// TIA Portal V16 export
// export: Created 2021-05-26T11:52:20.4679545Z, ExportSetting WithDefaults, DisplayName Totally Integrated Automation Portal, DisplayVersion V16 Update 4, DisplayName TIA Portal Version Control Interface, DisplayVersion V16 Update 2, DisplayName TIA Portal Openness, DisplayVersion V16 Update 4, DisplayName STEP 7 Professional, DisplayVersion V16 Update 4, DisplayName STEP 7 Safety, DisplayVersion V16, DisplayName WinCC Advanced, DisplayVersion V16 Update 4
DATA_BLOCK "DB_BC"   // DB10
{ S7_Optimized_Access := 'FALSE'; DB_Accessible_From_OPC_UA := 'FALSE' }
VERSION : 0.1
// stored: AutoNumber false, DBAccessibleFromOPCUA false, IsOnlyStoredInLoadMemory false, IsWriteProtectedInAS false
   VAR
      Spare0 : Byte;
      cmdRegLo : Bool;
      cmdBCRstHi : Bool;
      res_b1_2 : Bool;
      res_b1_3 : Bool;
      res_b1_4 : Bool;
      res_b1_5 : Bool;
      res_b1_6 : Bool;
      res_b1_7 : Bool;
      BC_TrigDelay : UInt;
      SwpStartTime : UInt;
      SwpTimeStep : UInt;
      sweepMod : Byte;
      CommCnt : Byte;
      res_b10 : Byte;
      res_b11 : Byte;
      stRfSwitch : Bool;
      stReflection : Bool;
      stRfEvent : Bool;
      stSumInterlock : Bool;
      stRfEnable : Bool;
      stTriggerBC : Bool;
      res_ib0_6 : Bool;
      res_ib0_7 : Bool;
      LatMPS_IL : Bool;
      LatTTL2 : Bool;
      LatTTL3 : Bool;
      LatTTL4 : Bool;
      LatRfAcdcBackDoor : Bool;
      LatRfFrontDoor : Bool;
      LatRectTmpSw : Bool;
      LatPhaseLoss : Bool;
      LatModConnect : Bool;
      LatModTmpSw : Bool;
      LatEmergency : Bool;
      LatmjCabinet : Bool;
      LatSafetyILck : Bool;
      LatCircArc : Bool;
      LatLoadArc : Bool;
      LatCavVac : Bool;
      stMPS_IL : Bool;
      stTTL2 : Bool;
      stTTL3 : Bool;
      stTTL4 : Bool;
      stRfAcdcBackDoor : Bool;
      stRfFrontDoor : Bool;
      RectTmpSw : Bool;
      PhaseLoss : Bool;
      ModConnect : Bool;
      ModTmpSw : Bool;
      Emergency : Bool;
      mjCabinet : Bool;
      SafetyILck : Bool;
      stCircArc : Bool;
      stLoadArc : Bool;
      stCavVac : Bool;
      stPinSSA : Bool;
      stPfrwPrDrv1 : Bool;
      stPfrwPrDrv2 : Bool;
      stRFSpare1 : Bool;
      stPfrwSsa : Bool;
      stPrflSsa : Bool;
      stPfrwDrv : Bool;
      stPrflDrv : Bool;
      stPrflMod1 : Bool;
      stPrflMod2 : Bool;
      stPrflMod3 : Bool;
      stPrflMod4 : Bool;
      stPrflMod5 : Bool;
      stPrflMod6 : Bool;
      stPrflMod7 : Bool;
      stPrflMod8 : Bool;
      stPrflMod9 : Bool;
      stPrflMod10 : Bool;
      stPrflMod11 : Bool;
      stPrflMod12 : Bool;
      stPrflMod13 : Bool;
      stPrflMod14 : Bool;
      stPrflMod15 : Bool;
      "stRFpare 2" : Bool;
      stPfrwMod1 : Bool;
      stPfrwMod2 : Bool;
      stPfrwMod3 : Bool;
      stPfrwMod4 : Bool;
      stPfrwMod5 : Bool;
      stPfrwMod6 : Bool;
      stPfrwMod7 : Bool;
      stPfrwMod8 : Bool;
      stPfrwMod9 : Bool;
      stPfrwMod10 : Bool;
      stPfrwMod11 : Bool;
      stPfrwMod12 : Bool;
      stPfrwMod13 : Bool;
      stPfrwMod14 : Bool;
      stPfrwMod15 : Bool;
      "stRFSpare 3" : Bool;
      stPfrwCircIn : Bool;
      stPrflCircIn : Bool;
      stPfrwCircOut : Bool;
      stPrflCircOut : Bool;
      stPfrwCircLoad : Bool;
      stPrflCircLoad : Bool;
      stPfrwCoupl : Bool;
      stPrflCoupl : Bool;
      SW_Version : Byte;
      PwrFrwSsa : Int;
      PwrRflSsa : Int;
      PwrPinSsa : Int;
      PwrFrwPrDrv1 : Int;
      PwrFrwPrDrv2 : Int;
      PwrFrwDrv : Int;
      PwrRflDrv : Int;
      PwrFrwMod1 : Int;
      PwrFrwMod2 : Int;
      PwrFrwMod3 : Int;
      PwrFrwMod4 : Int;
      PwrFrwMod5 : Int;
      PwrFrwMod6 : Int;
      PwrFrwMod7 : Int;
      PwrFrwMod8 : Int;
      PwrFrwMod9 : Int;
      PwrFrwMod10 : Int;
      PwrFrwMod11 : Int;
      PwrFrwMod12 : Int;
      PwrFrwMod13 : Int;
      PwrFrwMod14 : Int;
      PwrFrwMod15 : Int;
      PwrRflMod1 : Int;
      PwrRflMod2 : Int;
      PwrRflMod3 : Int;
      PwrRflMod4 : Int;
      PwrRflMod5 : Int;
      PwrRflMod6 : Int;
      PwrRflMod7 : Int;
      PwrRflMod8 : Int;
      PwrRflMod9 : Int;
      PwrRflMod10 : Int;
      PwrRflMod11 : Int;
      PwrRflMod12 : Int;
      PwrRflMod13 : Int;
      PwrRflMod14 : Int;
      PwrRflMod15 : Int;
      PfrwCircIn : Int;
      PrflCircIn : Int;
      PfrwCircOut : Int;
      PrflCircOut : Int;
      PfrwCircLoad : Int;
      PrflCircLoad : Int;
      PfrwCoupl : Int;
      PrflCoupl : Int;
      CommCnt_1 : Byte;
      swpPwrFrwSsa : "UDT_swp51Data";
      swpPwrRflSsa { S7_SetPoint := 'True'} : "UDT_swp51Data";
      swpPwrFrwMod { S7_SetPoint := 'True'} : "UDT_swp51Data";
      swpPwrRflMod { S7_SetPoint := 'True'} : "UDT_swp51Data";
      swpPwrPinSsa { S7_SetPoint := 'True'} : "UDT_swp51Data";
      CommCnt_2 : Byte;
   END_VAR
BEGIN
END_DATA_BLOCK
